// TIA Portal project "baicuoikiA+" (V15)

(* hardware
DEVICE "S7-1200 station_1"  S7-1200 Station
   slot 0: "Rack_0"  S7-1200 Rack  Rack  V1.0
   slot 1: "PLC_1"  CPU 1214C AC/DC/Rly  6ES7 214-1BG40-0XB0  V4.2
DEVICE "PC-System_1"  SIMATIC PC station
   slot 0: "SIMATIC PC station"  Rail  SIMATIC PC-Station  V1.0
      slot 125: "Stationmanager"  Station_Manager  V6.0.4
   slot 1: "HMI_RT_1"  WinCC RT Advanced  6AV2 104-0xxxx-xxxx  15.0.0.0
      slot 33792: "Host interface"  Host interface
   slot 2: "IE general_1"  IE General  IE_CP  V8.2.0
*)

// ===== PLC "PLC_1"  CPU 1214C AC/DC/Rly =====

VAR_GLOBAL   // PLC tag table "Default tag table"
   "Clock_Byte" AT %MB5 : Byte;
   "Clock_10Hz" AT %M5.0 : Bool;
   "Clock_5Hz" AT %M5.1 : Bool;
   "Clock_2.5Hz" AT %M5.2 : Bool;
   "Clock_2Hz" AT %M5.3 : Bool;
   "Clock_1.25Hz" AT %M5.4 : Bool;
   "Clock_1Hz" AT %M5.5 : Bool;
   "Clock_0.625Hz" AT %M5.6 : Bool;
   "Clock_0.5Hz" AT %M5.7 : Bool;
   "tag_1" AT %M50.0 : Bool;
   "tag_2" AT %M50.1 : Bool;
   "tag_3" AT %M50.2 : Bool;
   "tag_4" AT %M50.3 : Bool;
   "tag_5" AT %M50.4 : Bool;
   "tag_6" AT %M50.5 : Bool;
   "tag_7" AT %M50.6 : Bool;
   "tag_8" AT %M50.7 : Bool;
   "tag_9" AT %M51.0 : Bool;
   "tag_10" AT %M51.1 : Bool;
   "tag_11" AT %M51.2 : Bool;
   "tag_12" AT %M51.3 : Bool;
   "tag_13" AT %M51.4 : Bool;
   "tag_14" AT %M51.5 : Bool;
   "tag_15" AT %M51.6 : Bool;
   "tag_16" AT %M51.7 : Bool;
   "tag_17" AT %M52.0 : Bool;
   "tag_18" AT %M52.1 : Bool;
   "tag_19" AT %M52.2 : Bool;
   "tag_20" AT %M52.3 : Bool;
   "tag_21" AT %M52.4 : Bool;
   "tag_22" AT %M52.5 : Bool;
END_VAR

VAR_GLOBAL   // PLC tag table "Input"
   "Start" AT %M0.0 : Bool;
   "Stop" AT %M0.1 : Bool;
   "Select_Mode" AT %M0.2 : Bool;
   "Low_Sensor" AT %M0.3 : Bool;
   "Avg_Sensor" AT %M0.4 : Bool;
   "High_Sensor" AT %M0.5 : Bool;
   "Affix_Sensor" AT %M0.6 : Bool;
   "Reset_all" AT %M0.7 : Bool;
   "Reset_count" AT %M1.0 : Bool;
   "check_realtime" AT %M1.1 : Bool;
   "check_storage" AT %M1.2 : Bool;
   "Start_belt_main" AT %M1.3 : Bool;
   "Stop_belt_main" AT %M1.4 : Bool;
   "Start_belt_low" AT %M1.5 : Bool;
   "Start_belt_avg" AT %M1.6 : Bool;
   "Stop_belt_low" AT %M1.7 : Bool;
   "Stop_belt_lavg" AT %M2.0 : Bool;
   "Start_belt_high" AT %M2.1 : Bool;
   "Stop_belt_high" AT %M2.2 : Bool;
   "Start_affix_machine" AT %M2.3 : Bool;
   "Stop_affix_machine" AT %M2.4 : Bool;
   "Change_Pass" AT %M2.5 : Bool;
   "Reset_change_pass" AT %M2.6 : Bool;
END_VAR

VAR_GLOBAL   // PLC tag table "Output"
   "Belt_main" AT %Q0.0 : Bool;
   "Belt_Low_Product" AT %Q0.1 : Bool;
   "Belt_high_Product" AT %Q0.2 : Bool;
   "Xylanh_high_product" AT %Q0.3 : Bool;
   "Xylanh_low_prodcut" AT %Q0.4 : Bool;
   "Affix_machine" AT %Q0.5 : Bool;
   "Lamp_run_auto" AT %Q0.6 : Bool;
   "Lamp_run_manu" AT %Q0.7 : Bool;
   "Q_Low_sensor" AT %Q1.0 : Bool;
   "Q_avg_sensor" AT %Q1.1 : Bool;
   "Q-high_sensor" AT %Q1.2 : Bool;
   "Belt_avg_product" AT %Q1.3 : Bool;
END_VAR

VAR_GLOBAL   // PLC tag table "Tag_simu_count"
   "count_high_product" AT %MW10 : Int;
   "count_low_product" AT %MW12 : Int;
   "count_avg_product" AT %MW14 : Int;
   "count_all" AT %MW16 : Int;
   "Sim_front" AT %MW18 : Int;
   "Sim_back" AT %MW20 : Int;
   "Sim_belt_low" AT %MW22 : Int;
   "Sim_belt_avg" AT %MW24 : Int;
   "Sim_belt_high" AT %MW26 : Int;
   "Sim_xylanh_low" AT %MW28 : Int;
   "Sim_xylanh_avg" AT %MW32 : Int;
   "count_total_low" AT %MW34 : Int;
   "count_total_avg" AT %MW36 : Int;
   "count_total_high" AT %MW38 : Int;
   "count_box_low" AT %MW40 : Int;
   "count_box_avg" AT %MW42 : Int;
   "count_box_high" AT %MW44 : Int;
   "change_low" AT %MW46 : Int;
   "change_avg" AT %MW48 : Int;
   "chang_high" AT %MW54 : Int;
END_VAR

VAR_GLOBAL   // PLC tag table "Bit_trung_gian"
   "TG" AT %M30.0 : Bool;
   "TG_1" AT %M30.1 : Bool;
   "TG_2" AT %M30.2 : Bool;
   "TG_3" AT %M30.3 : Bool;
   "TG_4" AT %M30.4 : Bool;
   "TG_5" AT %M30.5 : Bool;
   "TG_6" AT %M30.6 : Bool;
   "TG_7" AT %M30.7 : Bool;
   "TG_8" AT %M31.0 : Bool;
   "TG_9" AT %M31.1 : Bool;
   "TG_10" AT %M31.2 : Bool;
   "TG_11" AT %M31.3 : Bool;
END_VAR

// folder: System blocks/Program resources

DATA_BLOCK "Ton_affix_machine"   // DB1
{ S7_Optimized_Access := 'TRUE' }
AUTHOR : Simatic
FAMILY : IEC
NAME : IEC_TMR
VERSION : 1.0
// stored: InstanceOfName IEC_TIMER
"IEC_TIMER"
BEGIN
END_DATA_BLOCK

DATA_BLOCK "Count_Low_Productt"   // DB2
{ S7_Optimized_Access := 'TRUE' }
AUTHOR : Simatic
FAMILY : IEC
NAME : CNTR
VERSION : 1.0
// stored: InstanceOfName IEC_COUNTER
"IEC_COUNTER"
BEGIN
END_DATA_BLOCK

DATA_BLOCK "Timer_reset_xylanh_low"   // DB3
{ S7_Optimized_Access := 'TRUE' }
AUTHOR : Simatic
FAMILY : IEC
NAME : IEC_TMR
VERSION : 1.0
// stored: InstanceOfName IEC_TIMER
"IEC_TIMER"
BEGIN
END_DATA_BLOCK

DATA_BLOCK "delay_sim_back"   // DB4
{ S7_Optimized_Access := 'TRUE' }
AUTHOR : Simatic
FAMILY : IEC
NAME : IEC_TMR
VERSION : 1.0
// stored: InstanceOfName IEC_TIMER
"IEC_TIMER"
BEGIN
END_DATA_BLOCK

DATA_BLOCK "Delay_belt_low"   // DB5
{ S7_Optimized_Access := 'TRUE' }
AUTHOR : Simatic
FAMILY : IEC
NAME : IEC_TMR
VERSION : 1.0
// stored: InstanceOfName IEC_TIMER
"IEC_TIMER"
BEGIN
END_DATA_BLOCK

DATA_BLOCK "Count_avg_Productt"   // DB6
{ S7_Optimized_Access := 'TRUE' }
AUTHOR : Simatic
FAMILY : IEC
NAME : CNTR
VERSION : 1.0
// stored: InstanceOfName IEC_COUNTER
"IEC_COUNTER"
BEGIN
END_DATA_BLOCK

DATA_BLOCK "Delay_belt_avg"   // DB7
{ S7_Optimized_Access := 'TRUE' }
AUTHOR : Simatic
FAMILY : IEC
NAME : IEC_TMR
VERSION : 1.0
// stored: InstanceOfName IEC_TIMER
"IEC_TIMER"
BEGIN
END_DATA_BLOCK

DATA_BLOCK "Timer_reset_xylanh_avg"   // DB8
{ S7_Optimized_Access := 'TRUE' }
AUTHOR : Simatic
FAMILY : IEC
NAME : IEC_TMR
VERSION : 1.0
// stored: InstanceOfName IEC_TIMER
"IEC_TIMER"
BEGIN
END_DATA_BLOCK

DATA_BLOCK "Count_high_Productt"   // DB9
{ S7_Optimized_Access := 'TRUE' }
AUTHOR : Simatic
FAMILY : IEC
NAME : CNTR
VERSION : 1.0
// stored: InstanceOfName IEC_COUNTER
"IEC_COUNTER"
BEGIN
END_DATA_BLOCK

DATA_BLOCK "Delay_belt_high"   // DB10
{ S7_Optimized_Access := 'TRUE' }
AUTHOR : Simatic
FAMILY : IEC
NAME : IEC_TMR
VERSION : 1.0
// stored: InstanceOfName IEC_TIMER
"IEC_TIMER"
BEGIN
END_DATA_BLOCK

// folder: (top level)

FUNCTION "Select_Program" : Void   // FC1, LAD
{ S7_Optimized_Access := 'TRUE' }
VERSION : 0.1
   VAR_TEMP   // added for the SCL form of the ladder/FBD networks
      _w1 : Bool;
   END_VAR
BEGIN

REGION Network 1
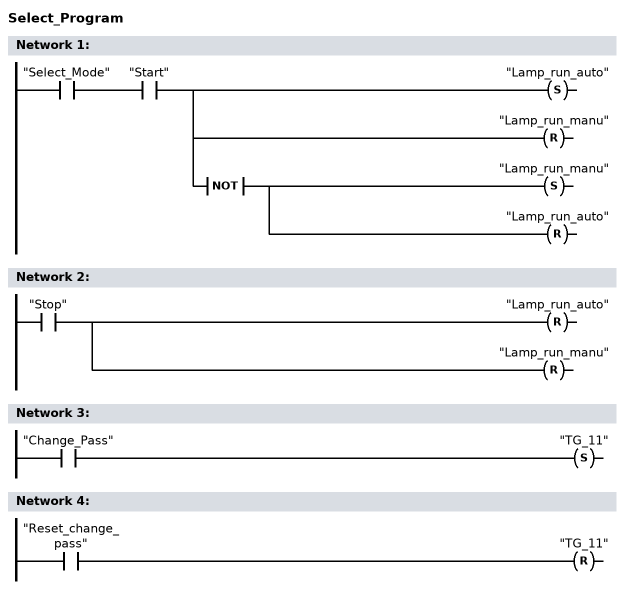
   RUNG wire#powerrail
      Contact( "Select_Mode" )
      Contact( "Start" )
      wire#w1
      S_Coil( "Lamp_run_auto" )
   END_RUNG
   RUNG wire#w1
      R_Coil( "Lamp_run_manu" )
   END_RUNG
   RUNG wire#w1
      Not()
      wire#w2
      S_Coil( "Lamp_run_manu" )
   END_RUNG
   RUNG wire#w2
      R_Coil( "Lamp_run_auto" )
   END_RUNG
   // the same network as SCL:
   #_w1 := "Select_Mode" AND "Start";
   IF #_w1 THEN
       "Lamp_run_auto" := TRUE;
       "Lamp_run_manu" := FALSE;
   END_IF;
   IF NOT #_w1 THEN
       "Lamp_run_manu" := TRUE;
       "Lamp_run_auto" := FALSE;
   END_IF;
END_REGION

REGION Network 2
   RUNG wire#powerrail
      Contact( "Stop" )
      wire#w1
      R_Coil( "Lamp_run_auto" )
   END_RUNG
   RUNG wire#w1
      R_Coil( "Lamp_run_manu" )
   END_RUNG
   // the same network as SCL:
   IF "Stop" THEN
       "Lamp_run_auto" := FALSE;
       "Lamp_run_manu" := FALSE;
   END_IF;
END_REGION

REGION Network 3
   RUNG wire#powerrail
      Contact( "Change_Pass" )
      S_Coil( "TG_11" )
   END_RUNG
   // the same network as SCL:
   IF "Change_Pass" THEN "TG_11" := TRUE; END_IF;
END_REGION

REGION Network 4
   RUNG wire#powerrail
      Contact( "Reset_change_pass" )
      R_Coil( "TG_11" )
   END_RUNG
   // the same network as SCL:
   IF "Reset_change_pass" THEN "TG_11" := FALSE; END_IF;
END_REGION
END_FUNCTION

FUNCTION "Auto_Program" : Void   // FC2, LAD
{ S7_Optimized_Access := 'TRUE' }
VERSION : 0.1
   VAR_TEMP   // added for the SCL form of the ladder/FBD networks
      _w1 : Bool;
      _w2 : Bool;
   END_VAR
BEGIN

REGION Network 1
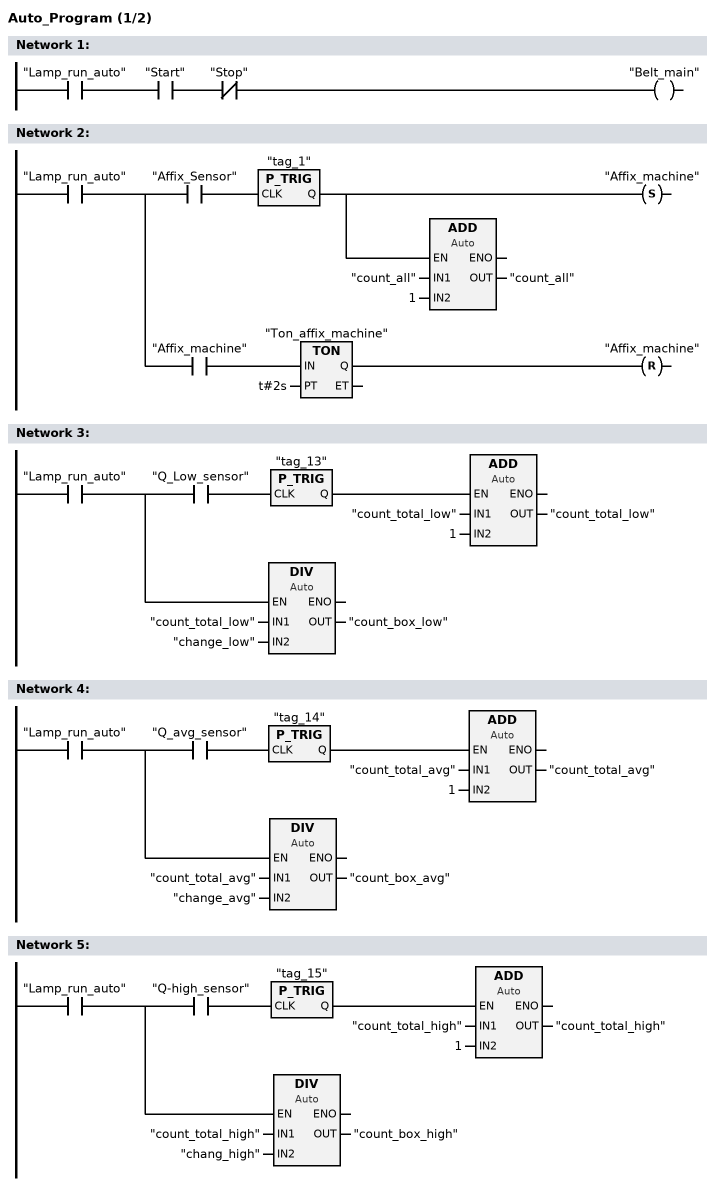
   RUNG wire#powerrail
      Contact( "Lamp_run_auto" )
      Contact( "Start" )
      I_Contact( "Stop" )
      Coil( "Belt_main" )
   END_RUNG
   // the same network as SCL:
   "Belt_main" := "Lamp_run_auto" AND "Start" AND NOT "Stop";
END_REGION

REGION Network 2
   #_w1 := "Lamp_run_auto" AND "Affix_Sensor";
   #_w2 := #_w1 AND NOT "tag_1";   // rising edge
   "tag_1" := #_w1;
   IF #_w2 THEN
       "Affix_machine" := TRUE;
       "count_all" := "count_all" + 1;
   END_IF;
   "Ton_affix_machine".TON(IN := "Lamp_run_auto" AND "Affix_machine", PT := t#2s);
   IF "Ton_affix_machine".Q THEN "Affix_machine" := FALSE; END_IF;
END_REGION

REGION Network 3
   RUNG wire#powerrail
      Contact( "Lamp_run_auto" )
      wire#w1
      Contact( "Q_Low_sensor" )
      P_Trig( "tag_13" )
      Add(in1 := "count_total_low", in2 := 1, out => "count_total_low")
   END_RUNG
   RUNG wire#w1
      Div(in1 := "count_total_low", in2 := "change_low", out => "count_box_low")
   END_RUNG
   // the same network as SCL:
   #_w1 := "Lamp_run_auto" AND "Q_Low_sensor";
   #_w2 := #_w1 AND NOT "tag_13";   // rising edge
   "tag_13" := #_w1;
   IF #_w2 THEN "count_total_low" := "count_total_low" + 1; END_IF;
   IF "Lamp_run_auto" THEN "count_box_low" := "count_total_low" / "change_low"; END_IF;
END_REGION

REGION Network 4
   RUNG wire#powerrail
      Contact( "Lamp_run_auto" )
      wire#w1
      Contact( "Q_avg_sensor" )
      P_Trig( "tag_14" )
      Add(in1 := "count_total_avg", in2 := 1, out => "count_total_avg")
   END_RUNG
   RUNG wire#w1
      Div(in1 := "count_total_avg", in2 := "change_avg", out => "count_box_avg")
   END_RUNG
   // the same network as SCL:
   #_w1 := "Lamp_run_auto" AND "Q_avg_sensor";
   #_w2 := #_w1 AND NOT "tag_14";   // rising edge
   "tag_14" := #_w1;
   IF #_w2 THEN "count_total_avg" := "count_total_avg" + 1; END_IF;
   IF "Lamp_run_auto" THEN "count_box_avg" := "count_total_avg" / "change_avg"; END_IF;
END_REGION

REGION Network 5
   RUNG wire#powerrail
      Contact( "Lamp_run_auto" )
      wire#w1
      Contact( "Q-high_sensor" )
      P_Trig( "tag_15" )
      Add(in1 := "count_total_high", in2 := 1, out => "count_total_high")
   END_RUNG
   RUNG wire#w1
      Div(in1 := "count_total_high", in2 := "chang_high", out => "count_box_high")
   END_RUNG
   // the same network as SCL:
   #_w1 := "Lamp_run_auto" AND "Q-high_sensor";
   #_w2 := #_w1 AND NOT "tag_15";   // rising edge
   "tag_15" := #_w1;
   IF #_w2 THEN "count_total_high" := "count_total_high" + 1; END_IF;
   IF "Lamp_run_auto" THEN "count_box_high" := "count_total_high" / "chang_high"; END_IF;
END_REGION

REGION Network 6
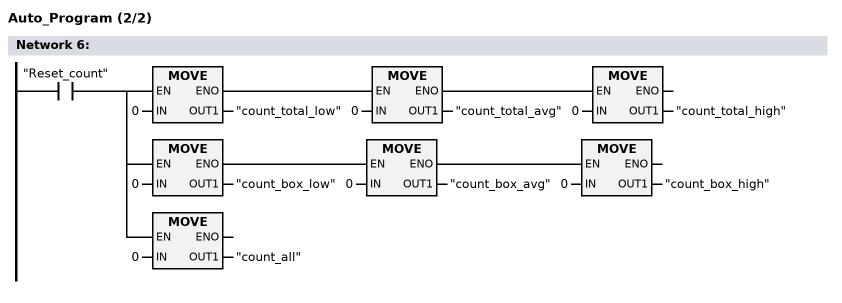
   RUNG wire#powerrail
      Contact( "Reset_count" )
      wire#w1
      Move(in := 0, out1 => "count_total_low")
      Move(in := 0, out1 => "count_total_avg")
      Move(in := 0, out1 => "count_total_high")
   END_RUNG
   RUNG wire#w1
      Move(in := 0, out1 => "count_box_low")
      Move(in := 0, out1 => "count_box_avg")
      Move(in := 0, out1 => "count_box_high")
   END_RUNG
   RUNG wire#w1
      Move(in := 0, out1 => "count_all")
   END_RUNG
   // the same network as SCL:
   IF "Reset_count" THEN
       "count_total_low" := 0;
       "count_total_avg" := 0;
       "count_total_high" := 0;
       "count_box_low" := 0;
       "count_box_avg" := 0;
       "count_box_high" := 0;
       "count_all" := 0;
   END_IF;
END_REGION
END_FUNCTION

FUNCTION "Manual_Program" : Void   // FC3, LAD
{ S7_Optimized_Access := 'TRUE' }
VERSION : 0.1
BEGIN

REGION Network 1
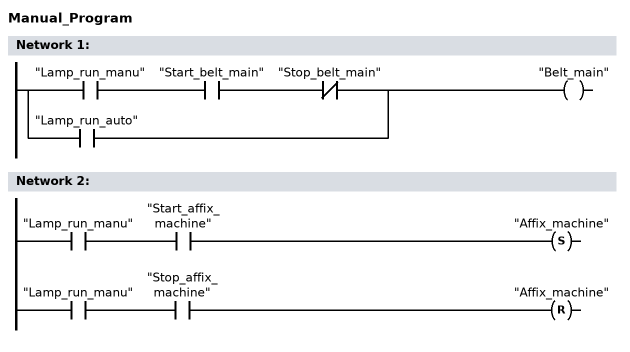
   RUNG wire#powerrail
      Contact( "Lamp_run_manu" )
      Contact( "Start_belt_main" )
      I_Contact( "Stop_belt_main" )
      wire#w1
      Coil( "Belt_main" )
   END_RUNG
   RUNG wire#powerrail
      Contact( "Lamp_run_auto" )
   END_RUNG wire#w1
   // the same network as SCL:
   "Belt_main" := ("Lamp_run_manu" AND "Start_belt_main" AND NOT "Stop_belt_main") OR "Lamp_run_auto";
END_REGION

REGION Network 2
   RUNG wire#powerrail
      Contact( "Lamp_run_manu" )
      Contact( "Start_affix_machine" )
      S_Coil( "Affix_machine" )
   END_RUNG
   RUNG wire#powerrail
      Contact( "Lamp_run_manu" )
      Contact( "Stop_affix_machine" )
      R_Coil( "Affix_machine" )
   END_RUNG
   // the same network as SCL:
   IF "Lamp_run_manu" AND "Start_affix_machine" THEN "Affix_machine" := TRUE; END_IF;
   IF "Lamp_run_manu" AND "Stop_affix_machine" THEN "Affix_machine" := FALSE; END_IF;
END_REGION
END_FUNCTION

FUNCTION "Simulation" : Void   // FC4, LAD
{ S7_Optimized_Access := 'TRUE' }
VERSION : 0.1
   VAR_TEMP   // added for the SCL form of the ladder/FBD networks
      _w1 : Bool;
      _w2 : Bool;
      _w3 : Bool;
      _w4 : Bool;
      _w5 : Bool;
   END_VAR
BEGIN

REGION Network 1: Block reset all
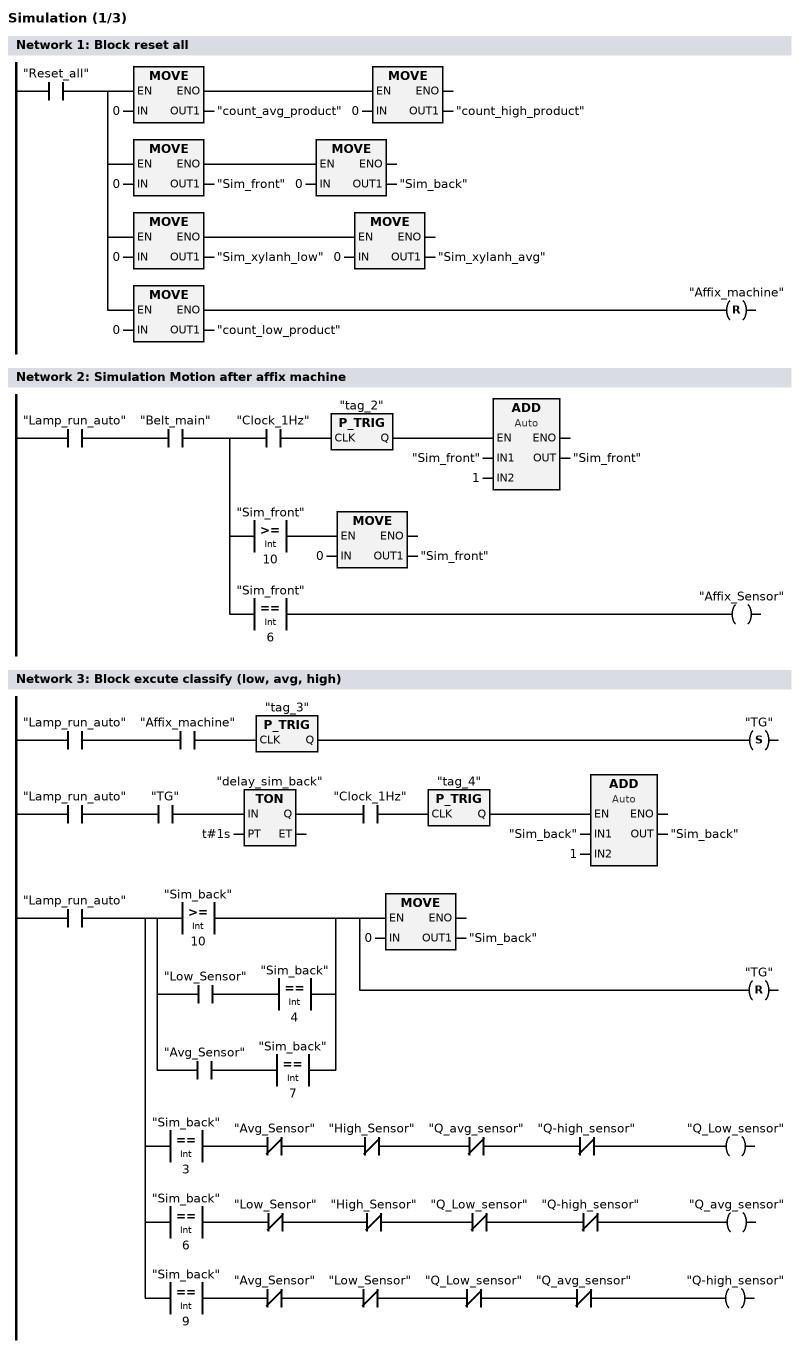
   RUNG wire#powerrail
      Contact( "Reset_all" )
      wire#w1
      Move(in := 0, out1 => "count_avg_product")
      Move(in := 0, out1 => "count_high_product")
   END_RUNG
   RUNG wire#w1
      Move(in := 0, out1 => "Sim_front")
      Move(in := 0, out1 => "Sim_back")
   END_RUNG
   RUNG wire#w1
      Move(in := 0, out1 => "Sim_xylanh_low")
      Move(in := 0, out1 => "Sim_xylanh_avg")
   END_RUNG
   RUNG wire#w1
      Move(in := 0, out1 => "count_low_product")
      R_Coil( "Affix_machine" )
   END_RUNG
   // the same network as SCL:
   IF "Reset_all" THEN
       "count_avg_product" := 0;
       "count_high_product" := 0;
       "Sim_front" := 0;
       "Sim_back" := 0;
       "Sim_xylanh_low" := 0;
       "Sim_xylanh_avg" := 0;
       "count_low_product" := 0;
       "Affix_machine" := FALSE;
   END_IF;
END_REGION

REGION Network 2: Simulation Motion after affix machine
   RUNG wire#powerrail
      Contact( "Lamp_run_auto" )
      Contact( "Belt_main" )
      wire#w1
      Contact( "Clock_1Hz" )
      P_Trig( "tag_2" )
      Add(in1 := "Sim_front", in2 := 1, out => "Sim_front")
   END_RUNG
   RUNG wire#w1
      { S7_Templates := "SrcType := Int" } GE_Contact(in1 := "Sim_front", in2 := 10)
      Move(in := 0, out1 => "Sim_front")
   END_RUNG
   RUNG wire#w1
      { S7_Templates := "SrcType := Int" } EQ_Contact(in1 := "Sim_front", in2 := 6)
      Coil( "Affix_Sensor" )
   END_RUNG
   // the same network as SCL:
   #_w1 := "Lamp_run_auto" AND "Belt_main";
   #_w2 := #_w1 AND "Clock_1Hz";
   #_w3 := #_w2 AND NOT "tag_2";   // rising edge
   "tag_2" := #_w2;
   IF #_w3 THEN "Sim_front" := "Sim_front" + 1; END_IF;
   IF #_w1 AND ("Sim_front" >= 10) THEN "Sim_front" := 0; END_IF;
   "Affix_Sensor" := #_w1 AND ("Sim_front" = 6);
END_REGION

REGION Network 3: Block excute classify (low, avg, high)
   #_w1 := "Lamp_run_auto" AND "Affix_machine";
   #_w2 := #_w1 AND NOT "tag_3";   // rising edge
   "tag_3" := #_w1;
   IF #_w2 THEN "TG" := TRUE; END_IF;
   "delay_sim_back".TON(IN := "Lamp_run_auto" AND "TG", PT := t#1s);
   #_w3 := "delay_sim_back".Q AND "Clock_1Hz";
   #_w4 := #_w3 AND NOT "tag_4";   // rising edge
   "tag_4" := #_w3;
   IF #_w4 THEN "Sim_back" := "Sim_back" + 1; END_IF;
   #_w5 := "Lamp_run_auto" AND (("Sim_back" >= 10) OR ("Low_Sensor" AND ("Sim_back" = 4)) OR ("Avg_Sensor" AND ("Sim_back" = 7)));
   IF #_w5 THEN
       "Sim_back" := 0;
       "TG" := FALSE;
   END_IF;
   "Q_Low_sensor" := "Lamp_run_auto" AND ("Sim_back" = 3) AND NOT "Avg_Sensor" AND NOT "High_Sensor" AND NOT "Q_avg_sensor" AND NOT "Q-high_sensor";
   "Q_avg_sensor" := "Lamp_run_auto" AND ("Sim_back" = 6) AND NOT "Low_Sensor" AND NOT "High_Sensor" AND NOT "Q_Low_sensor" AND NOT "Q-high_sensor";
   "Q-high_sensor" := "Lamp_run_auto" AND ("Sim_back" = 9) AND NOT "Avg_Sensor" AND NOT "Low_Sensor" AND NOT "Q_Low_sensor" AND NOT "Q_avg_sensor";
END_REGION

REGION Network 4
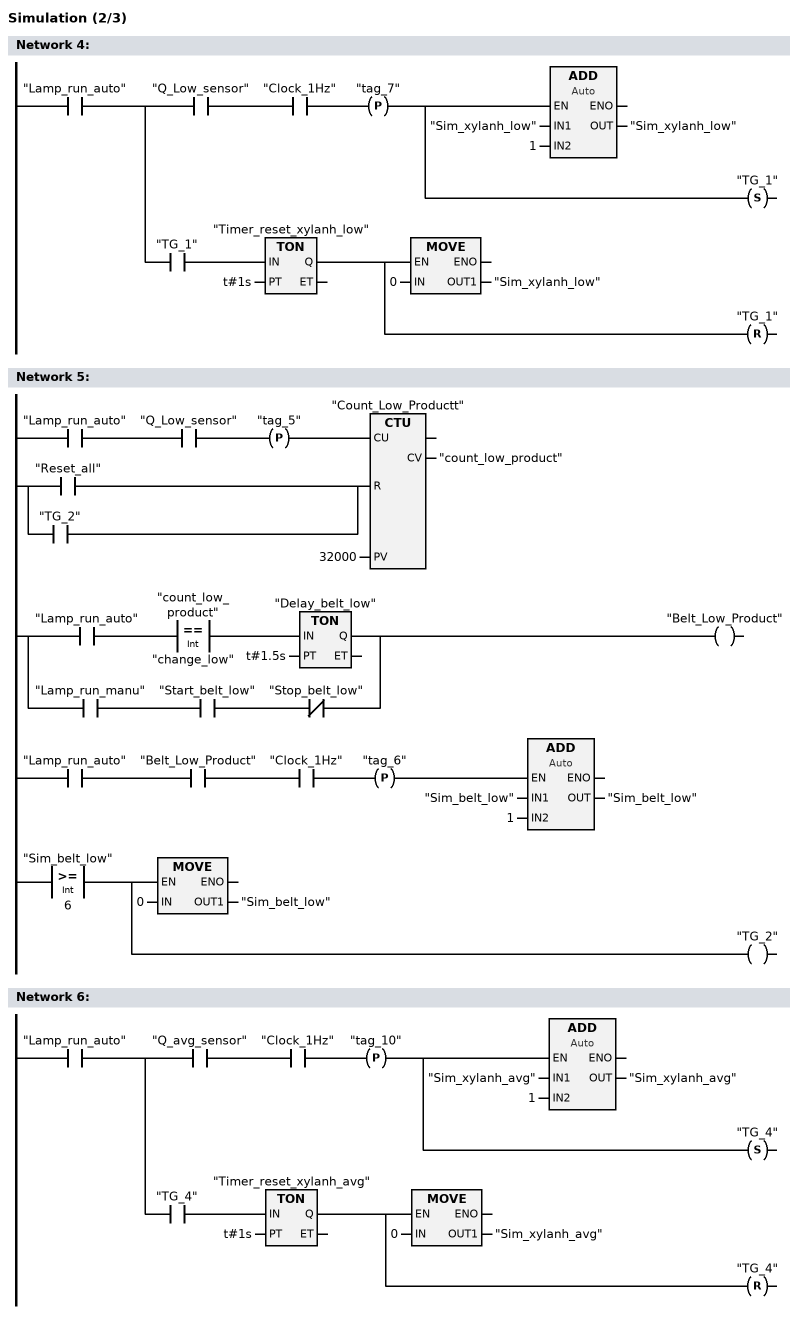
   #_w1 := "Lamp_run_auto" AND "Q_Low_sensor" AND "Clock_1Hz";
   #_w2 := #_w1 AND NOT "tag_7";   // rising edge
   "tag_7" := #_w1;
   IF #_w2 THEN
       "Sim_xylanh_low" := "Sim_xylanh_low" + 1;
       "TG_1" := TRUE;
   END_IF;
   "Timer_reset_xylanh_low".TON(IN := "Lamp_run_auto" AND "TG_1", PT := t#1s);
   IF "Timer_reset_xylanh_low".Q THEN
       "Sim_xylanh_low" := 0;
       "TG_1" := FALSE;
   END_IF;
END_REGION

REGION Network 5
   #_w1 := "Lamp_run_auto" AND "Q_Low_sensor";
   #_w2 := #_w1 AND NOT "tag_5";   // rising edge
   "tag_5" := #_w1;
   "Count_Low_Productt".CTU(CU := #_w2, R := "Reset_all" OR "TG_2", PV := 32000, CV => "count_low_product");
   "Delay_belt_low".TON(IN := "Lamp_run_auto" AND ("count_low_product" = "change_low"), PT := t#1.5s);
   "Belt_Low_Product" := "Delay_belt_low".Q OR ("Lamp_run_manu" AND "Start_belt_low" AND NOT "Stop_belt_low");
   #_w3 := "Lamp_run_auto" AND "Belt_Low_Product" AND "Clock_1Hz";
   #_w4 := #_w3 AND NOT "tag_6";   // rising edge
   "tag_6" := #_w3;
   IF #_w4 THEN "Sim_belt_low" := "Sim_belt_low" + 1; END_IF;
   #_w5 := "Sim_belt_low" >= 6;
   IF #_w5 THEN "Sim_belt_low" := 0; END_IF;
   "TG_2" := #_w5;
END_REGION

REGION Network 6
   #_w1 := "Lamp_run_auto" AND "Q_avg_sensor" AND "Clock_1Hz";
   #_w2 := #_w1 AND NOT "tag_10";   // rising edge
   "tag_10" := #_w1;
   IF #_w2 THEN
       "Sim_xylanh_avg" := "Sim_xylanh_avg" + 1;
       "TG_4" := TRUE;
   END_IF;
   "Timer_reset_xylanh_avg".TON(IN := "Lamp_run_auto" AND "TG_4", PT := t#1s);
   IF "Timer_reset_xylanh_avg".Q THEN
       "Sim_xylanh_avg" := 0;
       "TG_4" := FALSE;
   END_IF;
END_REGION

REGION Network 7
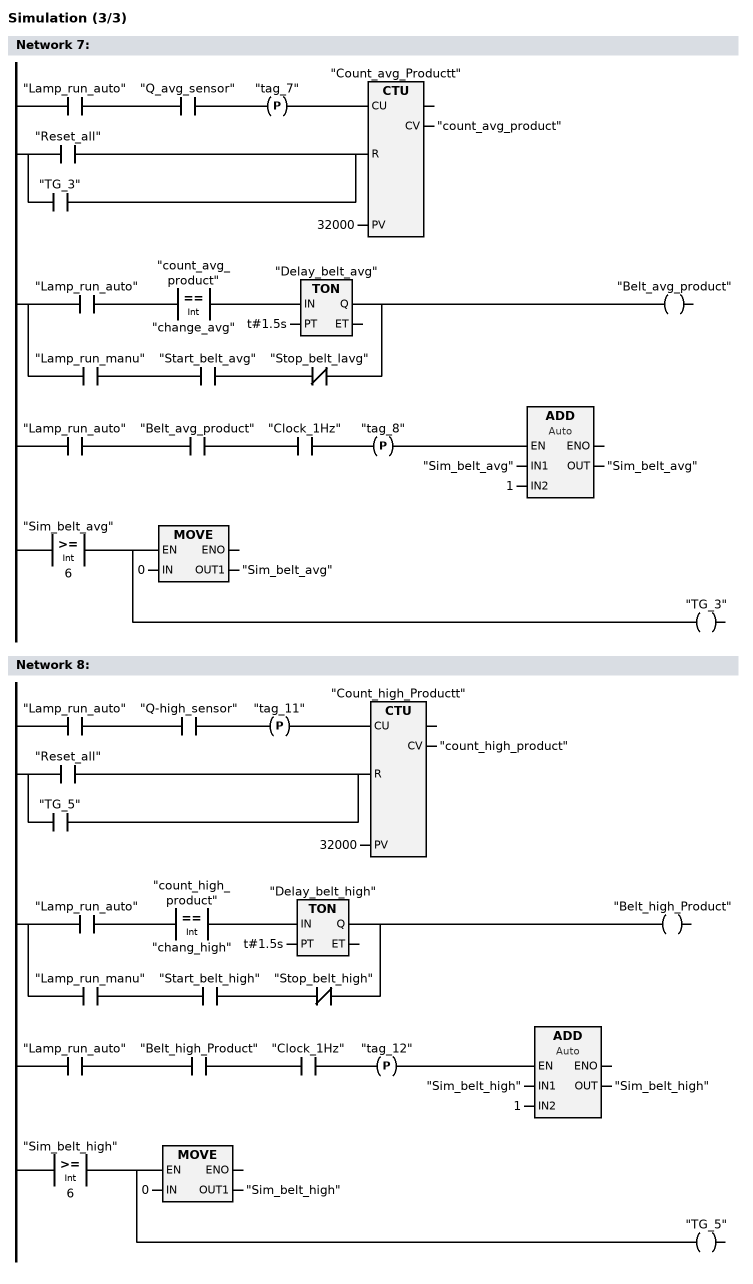
   #_w1 := "Lamp_run_auto" AND "Q_avg_sensor";
   #_w2 := #_w1 AND NOT "tag_7";   // rising edge
   "tag_7" := #_w1;
   "Count_avg_Productt".CTU(CU := #_w2, R := "Reset_all" OR "TG_3", PV := 32000, CV => "count_avg_product");
   "Delay_belt_avg".TON(IN := "Lamp_run_auto" AND ("count_avg_product" = "change_avg"), PT := t#1.5s);
   "Belt_avg_product" := "Delay_belt_avg".Q OR ("Lamp_run_manu" AND "Start_belt_avg" AND NOT "Stop_belt_lavg");
   #_w3 := "Lamp_run_auto" AND "Belt_avg_product" AND "Clock_1Hz";
   #_w4 := #_w3 AND NOT "tag_8";   // rising edge
   "tag_8" := #_w3;
   IF #_w4 THEN "Sim_belt_avg" := "Sim_belt_avg" + 1; END_IF;
   #_w5 := "Sim_belt_avg" >= 6;
   IF #_w5 THEN "Sim_belt_avg" := 0; END_IF;
   "TG_3" := #_w5;
END_REGION

REGION Network 8
   #_w1 := "Lamp_run_auto" AND "Q-high_sensor";
   #_w2 := #_w1 AND NOT "tag_11";   // rising edge
   "tag_11" := #_w1;
   "Count_high_Productt".CTU(CU := #_w2, R := "Reset_all" OR "TG_5", PV := 32000, CV => "count_high_product");
   "Delay_belt_high".TON(IN := "Lamp_run_auto" AND ("count_high_product" = "chang_high"), PT := t#1.5s);
   "Belt_high_Product" := "Delay_belt_high".Q OR ("Lamp_run_manu" AND "Start_belt_high" AND NOT "Stop_belt_high");
   #_w3 := "Lamp_run_auto" AND "Belt_high_Product" AND "Clock_1Hz";
   #_w4 := #_w3 AND NOT "tag_12";   // rising edge
   "tag_12" := #_w3;
   IF #_w4 THEN "Sim_belt_high" := "Sim_belt_high" + 1; END_IF;
   #_w5 := "Sim_belt_high" >= 6;
   IF #_w5 THEN "Sim_belt_high" := 0; END_IF;
   "TG_5" := #_w5;
END_REGION
END_FUNCTION

ORGANIZATION_BLOCK "Main"   // OB1, LAD, ProgramCycle
TITLE = "Main Program Sweep (Cycle)"
{ S7_Optimized_Access := 'TRUE' }
VERSION : 0.1
   VAR_INPUT
      Initial_Call : Bool;   // Initial call of this OB
      Remanence : Bool;   // =True, if remanent data are available
   END_VAR
BEGIN

REGION Network 1
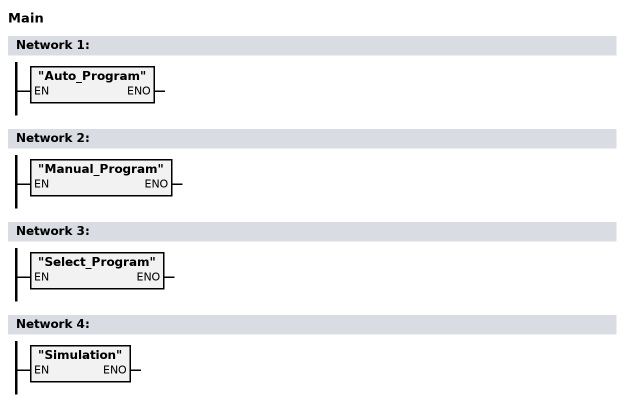
   RUNG wire#powerrail
      "Auto_Program"()
   END_RUNG
   // the same network as SCL:
   "Auto_Program"();
END_REGION

REGION Network 2
   RUNG wire#powerrail
      "Manual_Program"()
   END_RUNG
   // the same network as SCL:
   "Manual_Program"();
END_REGION

REGION Network 3
   RUNG wire#powerrail
      "Select_Program"()
   END_RUNG
   // the same network as SCL:
   "Select_Program"();
END_REGION

REGION Network 4
   RUNG wire#powerrail
      "Simulation"()
   END_RUNG
   // the same network as SCL:
   "Simulation"();
END_REGION
END_ORGANIZATION_BLOCK

(* ===== HMI "HMI_RT_1" =====
system functions are stored by id; their names below are inferred from use
connection "HMI_Connection_1": ETHERNET, S7_1200_OMS
connection "HMI_Connection_2": ETHERNET, S7_1200_OMS
connection "HMI_Connection_3": ETHERNET, S7_1200_OMS

HMI tags "Default tag table"
   "Sim_front" : Int = PLC Sim_front AT %MW18, 1 s
   "Lamp_run_auto" : Bool = PLC Lamp_run_auto AT %Q0.6, 1 s
   "Select_Mode" : Bool = PLC Select_Mode AT %M0.2, 1 s
   "Start" : Bool = PLC Start AT %M0.0, 1 s
   "Stop" : Bool = PLC Stop AT %M0.1, 1 s
   "Belt_main" : Bool = PLC Belt_main AT %Q0.0, 1 s
   "Sim_back" : Int = PLC Sim_back AT %MW20, 1 s
   "Affix_machine" : Bool = PLC Affix_machine AT %Q0.5, 1 s
   "Affix_Sensor" : Bool = PLC Affix_Sensor AT %M0.6, 1 s
   "Low_Sensor" : Bool = PLC Low_Sensor AT %M0.3, 1 s
   "Avg_Sensor" : Bool = PLC Avg_Sensor AT %M0.4, 1 s
   "High_Sensor" : Bool = PLC High_Sensor AT %M0.5, 1 s
   "Reset_all" : Bool = PLC Reset_all AT %M0.7, 1 s
   "Q_Low_sensor" : Bool = PLC Q_Low_sensor AT %Q1.0, 1 s
   "Q_avg_sensor" : Bool = PLC Q_avg_sensor AT %Q1.1, 1 s
   "Q-high_sensor" : Bool = PLC "Q-high_sensor" AT %Q1.2, 1 s
   "count_all" : Int = PLC count_all AT %MW16, 1 s
   "count_low_product" : Int = PLC count_low_product AT %MW12, 1 s
   "count_high_product" : Int = PLC count_high_product AT %MW10, 1 s
   "Sim_belt_low" : Int = PLC Sim_belt_low AT %MW22, 1 s
   "Sim_xylanh_low" : Int = PLC Sim_xylanh_low AT %MW28, 1 s
   "Sim_xylanh_avg" : Int = PLC Sim_xylanh_avg AT %MW32, 1 s
   "Belt_Low_Product" : Bool = PLC Belt_Low_Product AT %Q0.1, 1 s
   "Belt_avg_product" : Bool = PLC Belt_avg_product AT %Q1.3, 1 s
   "Sim_belt_avg" : Int = PLC Sim_belt_avg AT %MW24, 1 s
   "count_avg_product" : Int = PLC count_avg_product AT %MW14, 1 s
   "Belt_high_Product" : Bool = PLC Belt_high_Product AT %Q0.2, 1 s
   "Sim_belt_high" : Int = PLC Sim_belt_high AT %MW26, 1 s
   "Lamp_run_manu" : Bool = PLC Lamp_run_manu AT %Q0.7, 1 s
   "count_total_low" : Int = PLC count_total_low AT %MW34, 1 s
   "count_total_avg" : Int = PLC count_total_avg AT %MW36, 1 s
   "count_total_high" : Int = PLC count_total_high AT %MW38, 1 s
   "count_box_low" : Int = PLC count_box_low AT %MW40, 1 s
   "count_box_avg" : Int = PLC count_box_avg AT %MW42, 1 s
   "count_box_high" : Int = PLC count_box_high AT %MW44, 1 s
   "Reset_count" : Bool = PLC Reset_count AT %M1.0, 1 s
   "check_realtime" : Bool = PLC check_realtime AT %M1.1, 1 s
   "Start_belt_main" : Bool = PLC Start_belt_main AT %M1.3, 1 s
   "Stop_belt_main" : Bool = PLC Stop_belt_main AT %M1.4, 1 s
   "Start_belt_low" : Bool = PLC Start_belt_low AT %M1.5, 1 s
   "Stop_belt_low" : Bool = PLC Stop_belt_low AT %M1.7, 1 s
   "Start_belt_avg" : Bool = PLC Start_belt_avg AT %M1.6, 1 s
   "Stop_belt_lavg" : Bool = PLC Stop_belt_lavg AT %M2.0, 1 s
   "Start_belt_high" : Bool = PLC Start_belt_high AT %M2.1, 1 s
   "Stop_belt_high" : Bool = PLC Stop_belt_high AT %M2.2, 1 s
   "Start_affix_machine" : Bool = PLC Start_affix_machine AT %M2.3, 1 s
   "Stop_affix_machine" : Bool = PLC Stop_affix_machine AT %M2.4, 1 s
   "Username" : WString[50] AT %DB1.DBX0.0
   "change_low" : Int = PLC change_low AT %MW46, 1 s
   "change_avg" : Int = PLC change_avg AT %MW48, 1 s
   "chang_high" : Int = PLC chang_high AT %MW54, 1 s
   "TG_11" : Bool = PLC TG_11 AT %M31.3, 1 s
   "Change_Pass" : Bool = PLC Change_Pass AT %M2.5, 1 s
   "Reset_change_pass" : Bool = PLC Reset_change_pass AT %M2.6, 1 s

screen "Screen_2" 1920x1080
   SymbolLibrary "Symbol library_1" at 293,380 size 190x154
      Appearance <- "Affix_machine"
   SymbolLibrary "Symbol library_15" at 493,687 size 209x113
      Visibility <- "Belt_Low_Product"
   SymbolLibrary "Symbol library_20" at 421,414 size 51x112
      HorizontalMovement <- "Sim_back"
   TextField "Text field_1" at 427,467 size 34x22; Text 'TED'
   TextField "Text field_13" at 1491,67 size 119x22; Text 'Check Quantity'
   SymbolLibrary "Symbol library_25" at 1462,663 size 67x86
      Appearance <- "Belt_high_Product"
   SymbolLibrary "Symbol library_24" at 193,811 size 67x86
      Appearance <- "Belt_Low_Product"
   SymbolLibrary "Symbol library_10" at 1063,807 size 67x86
      Appearance <- "Belt_avg_product"
   SymbolLibrary "Symbol library_19" at 191,761 size 537x67
      Appearance <- "Belt_Low_Product"
   SymbolLibrary "Symbol library_18" at 692,752 size 508x74
      ProcessValue <- "Belt_avg_product"
      Appearance <- "Belt_avg_product"
   SymbolLibrary "Symbol library_12" at 1107,605 size 504x80
      ProcessValue <- "Belt_high_Product"
      Appearance <- "Belt_high_Product"
   SymbolLibrary "Symbol library_9" at 94,489 size 539x70
      Appearance <- "Belt_main"
   SymbolLibrary "Symbol library_2" at 364,267 size 52x88
      Appearance <- "Affix_Sensor"
   SymbolLibrary "Symbol library_3" at 1012,537 size 67x86
      Appearance <- "Belt_main"
   SymbolLibrary "Symbol library_8" at 669,299 size 31x103
      VerticalMovement <- "Sim_xylanh_low"
   SymbolLibrary "Symbol library_11" at 661,224 size 43x70
      Appearance <- "Q_Low_sensor"
   SymbolLibrary "Symbol library_13" at 896,228 size 45x68
      Appearance <- "Q_avg_sensor"
   SymbolLibrary "Symbol library_14" at 905,300 size 31x100
      VerticalMovement <- "Sim_xylanh_avg"
   SymbolLibrary "Symbol library_17" at 1128,330 size 47x78
      Appearance <- "Q-high_sensor"
   IOField "I/O field_1" at 502,862 size 73x39; FormatPattern 99999
      ProcessValue <- "count_low_product"
   IOField "I/O field_2" at 764,866 size 71x37; FormatPattern 99999
      ProcessValue <- "count_avg_product"
   IOField "I/O field_3" at 1491,482 size 69x38; FormatPattern 99999
      ProcessValue <- "count_high_product"
   IOField "I/O field_4" at 1509,307 size 77x43; FormatPattern 999999
      ProcessValue <- "count_all"
   Switch "Switch_1" at 65,75 size 153x65; CaptionText 'Select Mode'; TextOff 'MANUAL'; TextOn 'AUTO'
      on SwitchOn: SetBit("Select_Mode")
      on SwitchOff: ResetBit("Select_Mode")
      ProcessValue <- "Select_Mode"
   Button "Button_3" at 80,330 size 105x51; TextOff 'Reset system'
      on Press: SetBit("Reset_all")
      on Release: ResetBit("Reset_all")
   SymbolLibrary "Symbol library_21" at 152,424 size 51x95
      HorizontalMovement <- "Sim_front"
   Switch "Switch_2" at 43,665 size 89x53; CaptionText 'Low_Sensor'; TextOff 'OFF'; TextOn 'ON'
      on SwitchOn: SetBit("Low_Sensor")
      on SwitchOff: ResetBit("Low_Sensor")
   Switch "Switch_3" at 42,725 size 90x52; TextOn 'ON'; CaptionText 'Avg_Sensor'; TextOff 'OFF'
      on SwitchOff: ResetBit("Avg_Sensor")
      on SwitchOn: SetBit("Avg_Sensor")
   Switch "Switch_4" at 42,789 size 89x53; TextOn 'ON'; CaptionText 'High_Sensor'; TextOff 'OFF'
      on SwitchOff: ResetBit("High_Sensor")
      on SwitchOn: SetBit("High_Sensor")
   SymbolLibrary "Symbol library_4" at 432,489 size 477x70
      Appearance <- "Belt_main"
   SymbolLibrary "Symbol library_5" at 770,489 size 424x70
      Appearance <- "Belt_main"
   Group "Group" at 421,414 size 51x112
   SymbolLibrary "Symbol library_7" at 534,690 size 125x114
      HorizontalMovement <- "Sim_belt_low"
      Visibility <- "Belt_Low_Product"
   SymbolLibrary "Symbol library_22" at 796,680 size 125x114
      Visibility <- "Belt_avg_product"
      HorizontalMovement <- "Sim_belt_avg"
   SymbolLibrary "Symbol library_16" at 754,680 size 208x109
      Visibility <- "Belt_avg_product"
   SymbolLibrary "Symbol library_23" at 1157,542 size 125x114
      Visibility <- "Belt_high_Product"
      ProcessValue <- "Sim_belt_high"
      HorizontalMovement <- "Sim_belt_high"
   SymbolLibrary "Symbol library_6" at 1120,534 size 197x120
      Visibility <- "Belt_high_Product"
   TextField "Text field_2" at 16,641 size 145x22; Text 'Simulation_sensor'
   Switch "Switch_5" at 22,240 size 106x66; CaptionText 'Start'; TextOff 'OFF'; TextOn 'ON'
      on SwitchOn: SetBit("Start")
      on SwitchOff: ResetBit("Start")
   Switch "Switch_6" at 149,240 size 104x66; TextOn 'ON'; CaptionText 'Stop'; TextOff 'OFF'
      on SwitchOff: ResetBit("Stop")
      on SwitchOn: SetBit("Stop")
   TextField "Text field_3" at 459,835 size 162x22; Text 'Quantity low product'
   TextField "Text field_4" at 717,836 size 162x22; Text 'Quantity avg product'
   TextField "Text field_5" at 1439,455 size 167x22; Text 'Quantity high product'
   TextField "Text field_6" at 340,237 size 97x22; Text 'Affix Sensor'
      Appearance <- "Affix_Sensor"
   TextField "Text field_7" at 710,267 size 92x22; Text 'Low Sensor'
      Appearance <- "Low_Sensor"
   TextField "Text field_8" at 948,267 size 89x22; Text 'Avg Sensor'
      Appearance <- "Avg_Sensor"
   TextField "Text field_9" at 1174,359 size 95x22; Text 'High Sensor'
      Appearance <- "High_Sensor"
   Circle "Circle_1" at 29,156 size 69x69
      Appearance <- "Lamp_run_auto"
   TextField "Text field_10" at 44,179 size 39x22; Text 'Auto'
   Circle "Circle_2" at 181,160 size 65x65
      Appearance <- "Lamp_run_manu"
   TextField "Text field_11" at 185,179 size 59x22; Text 'Manual'
   TextField "Text field_12" at 1491,281 size 105x22; Text 'Total Product'
      Appearance <- "High_Sensor"
   IOField "I/O field_5" at 1402,143 size 77x43; FormatPattern 999999
      ProcessValue <- "count_total_low"
   TextField "Text field_14" at 1402,108 size 78x22; Text 'Total Low'
   IOField "I/O field_6" at 1509,143 size 77x43; FormatPattern 999999
      ProcessValue <- "count_total_avg"
   TextField "Text field_15" at 1511,108 size 75x22; Text 'Total Avg'
   IOField "I/O field_7" at 1614,143 size 77x43; FormatPattern 999999
      ProcessValue <- "count_total_high"
   TextField "Text field_16" at 1610,108 size 81x22; Text 'Total High'
   Group "Group_1" at 1480,56 size 139x44
   TextField "Text field_20" at 333,453 size 112x22; Text 'Lable machine'
      Visibility <- "Start"
   IOField "I/O field_8" at 1404,228 size 77x43; FormatPattern 999999
      ProcessValue <- "count_box_low"
   IOField "I/O field_9" at 1509,228 size 77x43; FormatPattern 999999
      ProcessValue <- "count_box_avg"
   IOField "I/O field_10" at 1614,228 size 77x43; FormatPattern 999999
      ProcessValue <- "count_box_high"
   TextField "Text field_21" at 1494,194 size 102x22; Text 'Quantity Box'
   Button "Button_1" at 1511,359 size 69x41; TextOff 'Reset'
      on Press: SetBit("Reset_count")
      on Release: ResetBit("Reset_count")
   TrendView "Trend view_1" at 1210,690 size 695x335
      Visibility <- "check_realtime"
   Button "Button_4" at 1590,356 size 117x43; TextOff 'Check strorage'
      on Press: ActivateScreen("Screen_3", 0)
   Switch "Switch_7" at 1396,342 size 108x61; CaptionText 'Trend Realtime'; TextOff 'OFF'; TextOn 'VIEW'
      on SwitchOn: SetBit("check_realtime")
      on SwitchOff: ResetBit("check_realtime")
   Switch "Switch_8" at 94,559 size 97x58; CaptionText 'Belt Main'; TextOff 'OFF'; TextOn 'ON'
      Visibility <- "Lamp_run_manu"
      on SwitchOn: SetBit("Start_belt_main"); ResetBit("Stop_belt_main")
      on SwitchOff: SetBit("Stop_belt_main"); ResetBit("Start_belt_main")
   AlarmView "Alarm view_1" at 377,35 size 878x142
   Switch "Switch_9" at 473,330 size 91x56; TextOn 'ON'; CaptionText 'Label Machine'; TextOff 'OFF'
      Visibility <- "Lamp_run_manu"
      on SwitchOn: SetBit("Start_affix_machine"); ResetBit("Stop_affix_machine")
      on SwitchOff: SetBit("Stop_affix_machine"); ResetBit("Start_affix_machine")
   Switch "Switch_10" at 272,843 size 97x58; TextOn 'ON'; CaptionText 'Low Belt'; TextOff 'OFF'
      Visibility <- "Lamp_run_manu"
      on SwitchOn: SetBit("Start_belt_low"); ResetBit("Stop_belt_low")
      on SwitchOff: SetBit("Stop_belt_low"); ResetBit("Start_belt_low")
   Switch "Switch_11" at 960,835 size 97x58; TextOn 'ON'; CaptionText 'Avg Belt'; TextOff 'OFF'
      Visibility <- "Lamp_run_manu"
      on SwitchOn: SetBit("Start_belt_avg"); ResetBit("Stop_belt_lavg")
      on SwitchOff: SetBit("Stop_belt_lavg"); ResetBit("Start_belt_avg")
   Switch "Switch_12" at 1614,583 size 97x58; TextOn 'ON'; CaptionText 'High Belt'; TextOff 'OFF'
      Visibility <- "Lamp_run_manu"
      on SwitchOn: SetBit("Start_belt_high"); ResetBit("Stop_belt_high")
      on SwitchOff: SetBit("Stop_belt_high"); ResetBit("Start_belt_high")
   Group "Group_3" at 564,556 size 172x117
   Group "Group_4" at 803,556 size 172x117
   Button "Button_2" at 1051,1002 size 96x32; TextOff 'Text'
      on Press: "VBFunction_1"()
   Button "Button_5" at 12,16 size 112x40; TextOff 'Back Screen1'
      on Press: ActivateScreen("Screen_1", 0)
   IOField "I/O field_11" at 503,936 size 73x39; Authorization "change"; FormatPattern 99999
      ProcessValue <- "change_low"
   TextField "Text field_17" at 485,907 size 110x22; Text 'Type Quantity'
   IOField "I/O field_12" at 764,938 size 73x39; Authorization "change"; FormatPattern 99999
      ProcessValue <- "change_avg"
   TextField "Text field_18" at 739,910 size 110x22; Text 'Type Quantity'
   IOField "I/O field_13" at 1491,550 size 73x36; Authorization "change"; FormatPattern 99999
      ProcessValue <- "chang_high"
   TextField "Text field_19" at 1448,526 size 146x22; Text 'Type Quantity high'

screen "Screen_3" 1920x1080
   TrendView "Trend view_1" at 18,105 size 873x751
   Button "Button_1" at 47,30 size 136x48; TextOff 'Back to Screen 2'
      on Press: ActivateScreen("Screen_2", 0)
   AlarmView "Alarm view_1" at 948,105 size 936x753

screen "Screen_1" 1920x1080
   TextField "Text field_17" at 437,26 size 636x50; Text 'PRODUCT LABELING, CLASSIFICATION AND PACKAGING SYSTEM'
   TextField "Text field_18" at 599,97 size 305x22; Text 'Name student: Ngô Đức Nam-20021164'
   TextField "Text field_19" at 645,125 size 217x22; Text 'Teacher: Nguyễn Quang Nhã'
   Button "Button_1" at 541,276 size 101x42; TextOff 'Login'
      on Press: function_a2a04561()
   Group "Group_2" at 399,26 size 720x137
   Button "Button_2" at 886,277 size 98x42; TextOff 'Logout'
      on Press: function_f23ef4c9(); SetBit("Reset_change_pass"); ResetBit("Change_Pass")
   IOField "I/O field_1" at 682,307 size 150x43; FormatPattern ??????????????????????????????????????????????????
      ProcessValue <- "Username"
   Button "Button_3" at 887,343 size 97x42; TextOff 'Enter'; Authorization "excute"
      on Press: ActivateScreen("Screen_2", 0)
   TextField "Text field_1" at 693,281 size 141x22; Text 'Current Username'
   UserView "User view_2" at 521,403 size 480x240
   UserView "User view_1" at 523,403 size 480x240
      Visibility <- "TG_11"
   Button "Button_4" at 541,343 size 101x42; TextOff 'Change Pass'; Authorization "change"
      on Press: SetBit("Change_Pass"); ResetBit("Reset_change_pass")

VB script "VBFunction_1"
   	Dim objShell
       Set objShell = CreateObject("WScript.Shell")
       Dim pythonExe, pythonScript
       pythonExe = "C:/Program Files/Python311/python.exe"
      	pythonScript = "D:\Project_Python\SCADA_GET_DATA\scada.py" 
       objShell.Run pythonExe & " " & pythonScript
       Set objShell = Nothing

scheduled task "showuserlogin"
   on Action: function_f41c6f6c("Username")
*)